// ---------------------------------------------------------------------------
// GLOBAL DATA BLOCK: _Ec
// Purpose: Stores and manages the state and structure of all registered entities 
//          and tracks the current scope under construction.

// This attribute ensures variables are accessed using qualified names (e.g., _Ec.iFirst)
{attribute 'qualified_only'}

VAR_GLOBAL INTERNAL    
    // Reference to the first registered entity in the global entity list
    iFirst: I_EntityNode;

    // Reference to the last registered entity in the global entity list
    iLast: I_EntityNode;

    // Points to the entity currently being constructed
    // Used to add components or nested entities during initialization
    iUnderConstruction: I_EntityNode;

    // Tracks how many nested entity scopes are currently under construction
    // Used to manage hierarchical or recursive construction logic
    nConstructedScopes: UDINT;
END_VAR

(* stored: Version 1.1.0.1
   GVL _Ec: Id {25f16a6e-7888-4e3e-877d-3b7e2fe9f871} *)
